{attribute addProperty BoxType "EJ3202-0000-0019"}
{attribute addProperty Id "RTD_Inputs_ChannelAT %I*ARRAY[0..2] OF RTD_Inputs_Channel_5763EEB96480WcStateAT %I*WcState_98A4DF7520.250InfoDataAT %I*InfoData_BC63D37F80100"}
{attribute addProperty CRC "2714103225"}
{attribute addProperty SizeInBites "146"}
{attribute addProperty SizeInBytes "18.25"}
TYPE EJ3202_559337F5 :
STRUCT
	{attribute addProperty Name "RTD_Inputs_Channel"}
	RTD_Inputs_Channel : ARRAY[0..2] OF RTD_Inputs_Channel_5763EEB9;
	{attribute addProperty Name "WcState"}
	WcState : WcState_98A4DF75;
	{attribute addProperty Name "InfoData"}
	InfoData : InfoData_BC63D37F;
END_STRUCT
END_TYPE

(* stored: Version 1.2.0.0, ProductVersion 3.1.4024.9
   DUT EJ3202_559337F5: Id {2e5f6db6-ee81-473f-8a39-3fe7be90f9e3} *)
